(* CoDeSys 2.3.9.47 project: staircase.pro *)
(* Libraries: Nexgenie.lib 28.8.18 12:27:24, Standard.lib 28.8.18 12:27:25, Nexgenie_Util.lib 28.8.18 12:27:24, Nexgenie_H.lib 28.8.18 12:27:24, VAW.lib 28.8.18 12:27:25, Modbus.lib 28.8.18 12:27:24 *)

(* PLC configuration (modules and I/O channels)
Nexgenie1000 [Root] node -1, in %IB0 out %QB0
  Nexgenie [Nexgenie] node 0, in %IB0 out %QB0
*)

(* POU PLC_PRG, LD *)
PROGRAM PLC_PRG
VAR
	A AT %IX0.0: BOOL;
	B AT %IX0.1: BOOL;
	X AT %QX0.0: BOOL;
END_VAR
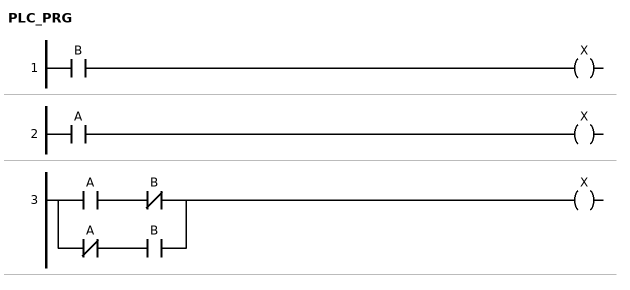
_LD_ (* Ladder Diagram *)
NETWORK 1
	[B] --- (X)
NETWORK 2
	[A] --- (X)
NETWORK 3
	{ [A] - [/B] | [/A] - [B] } --- (X)
_END_LD_
(* the same logic as Structured Text *)
(* Network 1 *)
X := B;
(* Network 2 *)
X := A;
(* Network 3 *)
X := A AND NOT B OR NOT A AND B;
END_PROGRAM

(* Visualisation LOL123
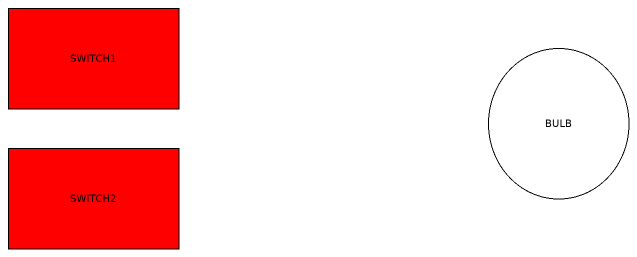
rectangle at (90,60)-(261,161): text "SWITCH1"; alarm colour if PLC_PRG.A; toggles PLC_PRG.A
rectangle at (90,200)-(261,301): text "SWITCH2"; alarm colour if PLC_PRG.B; toggles PLC_PRG.B
ellipse at (570,100)-(711,251): text "BULB"; alarm colour if PLC_PRG.X
*)
